Fanuc KAREL source: compact_preamble.KL

PROGRAM KT00096
%NOLOCKGROUP
VAR
H1 : ARRAY[2] OF SHORT
H2 : ARRAY[2] OF SHORT
OUT:REAL
BEGIN
H1[1]=2
H2[1]=3
H1[1]=2
H2[1]=3
OUT=((H1[1] * H2[1]))
END KT00096
